(* IEC 61131-3 sources: std_i2980_v2.06_cp053/Source/IMM/ieccontrol/TIG, 14 files *)

(* ---- FArraySum.pu ---- *)
(*
@h    ! WARNING !
@h    The Kemro K2 system (including software) only meets category B according to EN 954-1,
@h    thus it is not intended for usage in safety-relevant control applications in the field
@h    of personal safety (e.g. emergency stop).
@h    To implement potentially necessary safety-relevant control tasks, always use additional
@h    external safety devices that are intended for the particular purpose, and meet the necessary
@h    functional safety.
@h    For further information see EN 954-1 (EN ISO 13849-1) and/or the K2-x00 user manual, chapter
@h    "CE conformity, directives and standards".

calculates sum of n arrayelements of type DINT
*)

IMPORT_OVER_LISTFILE
 tyTIGDInt

END_IMPORT

FUNCTION FArraySum : DINT #DUMMY_EDIT_BLOCK

VAR_INPUT
 iNumber : DINT (* number of array elements *);
END_VAR

VAR_IN_OUT
 array : tyTIGDInt (* array *);
END_VAR

VAR
 tmpSum : DINT;
 i : DINT;
END_VAR
#BEGIN_EDIT_BLOCK
(**************************************** WARNING ********************************************
 *** The KEBA Kemro K2 System including software is not intended for safety control tasks! ***
 ***                       For further information see Comment tab!                        ***
 *********************************************************************************************)

tmpSum := 0;

FOR i := 1 TO iNumber DO
   tmpSum := tmpSum + array[i];
END_FOR;

FArraySum:= tmpSum;

;#END_EDIT_BLOCK END_FUNCTION

#END_OF_IEC_PART

@Puma @IecEditor 6 60 @Pou 25
@@@BEG_Comment@@@
@h    ! WARNING !
@h    The Kemro K2 system (including software) only meets category B according to EN 954-1,
@h    thus it is not intended for usage in safety-relevant control applications in the field
@h    of personal safety (e.g. emergency stop).
@h    To implement potentially necessary safety-relevant control tasks, always use additional
@h    external safety devices that are intended for the particular purpose, and meet the necessary
@h    functional safety.
@h    For further information see EN 954-1 (EN ISO 13849-1) and/or the K2-x00 user manual, chapter
@h    "CE conformity, directives and standards".

calculates sum of n arrayelements of type DINT
@@@END_Comment@@@

@BEG_Contents

@BEG_Func
@RT(17)FuncTreeContainer
0
@END_Func

@BEG_Const
@RT(18)ConstTreeContainer
0
@END_Const

@BEG_Export

@BEG_Kind
@FUNCTION @RT(9)FArraySum @STRUCTURED_TEXT
@RT(4)DINT @RT(0) @RT(0)
@END_Kind

@BEG_Dcl
@RT(16)DclTreeContainer
4
@Var @RT(7)iNumber @RT(0) @T @F @DT @RT(4)DINT @RT(0) @T @T @BASIC 0 @F
@F @F
@T
@BEG_Attrib
3 @RT(0) @RT(24)number of array elements @RT(0)
@END_Attrib
1 1 @F @F @F @F

@Var @RT(5)array @RT(0) @T @T @DERIVED 0 @T @T @DT @RT(9)tyTIGDInt @RT(0) @T @T @UNKNOWN 0 @F
@F @F
@T
@BEG_Attrib
3 @RT(0) @RT(5)array @RT(0)
@END_Attrib
1 2 @F @F @F @F

@Var @RT(6)tmpSum @RT(0) @T @F @DT @RT(4)DINT @RT(0) @T @T @BASIC 0 @F
@F @F
@T
@BEG_Attrib
3 @RT(0) @RT(0) @RT(0)
@END_Attrib
1 0 @F @F @F @F

@Var @RT(1)i @RT(0) @T @F @DT @RT(4)DINT @RT(0) @T @T @BASIC 0 @F
@F @F
@T
@BEG_Attrib
3 @RT(0) @RT(0) @RT(0)
@END_Attrib
1 0 @F @F @F @F

@END_Dcl

@END_Export

@BEG_Body
@TL(13)
(**************************************** WARNING ********************************************
 *** The KEBA Kemro K2 System including software is not intended for safety control tasks! ***
 ***                       For further information see Comment tab!                        ***
 *********************************************************************************************)

tmpSum := 0;

FOR i := 1 TO iNumber DO
   tmpSum := tmpSum + array[i];
END_FOR;

FArraySum:= tmpSum;

@END_Body

@END_Contents

(* ---- FDeleteActDSFiles.pu ---- *)
(*
@h    ! WARNING !
@h    The Kemro K2 system (including software) only meets category B according to EN 954-1,
@h    thus it is not intended for usage in safety-relevant control applications in the field
@h    of personal safety (e.g. emergency stop).
@h    To implement potentially necessary safety-relevant control tasks, always use additional
@h    external safety devices that are intended for the particular purpose, and meet the necessary
@h    functional safety.
@h    For further information see EN 954-1 (EN ISO 13849-1) and/or the K2-x00 user manual, chapter
@h    "CE conformity, directives and standards".

deletes and creates temporary directory for datasettransfer to tig

@FunctionID: A-VAR-14
@FunctionID: A-VAR-15
TIG 3.10
*)

IMPORT_OVER_LISTFILE
 KFILE_Status

END_IMPORT

FUNCTION FDeleteActDSFiles : BOOL #DUMMY_EDIT_BLOCK

VAR_IN_OUT
 sPath : STRING(255);
END_VAR

VAR
 s : KFILE_Status;
END_VAR
#BEGIN_EDIT_BLOCK
(**************************************** WARNING ********************************************
 *** The KEBA Kemro K2 System including software is not intended for safety control tasks! ***
 ***                       For further information see Comment tab!                        ***
 *********************************************************************************************)

s := KFILE_RemoveDir(sPath);
s := KFILE_MakeDir(sPath);
FDeleteActDSFiles := TRUE;

;#END_EDIT_BLOCK END_FUNCTION

#END_OF_IEC_PART

@Puma @IecEditor 6 60 @Pou 25
@@@BEG_Comment@@@
@h    ! WARNING !
@h    The Kemro K2 system (including software) only meets category B according to EN 954-1,
@h    thus it is not intended for usage in safety-relevant control applications in the field
@h    of personal safety (e.g. emergency stop).
@h    To implement potentially necessary safety-relevant control tasks, always use additional
@h    external safety devices that are intended for the particular purpose, and meet the necessary
@h    functional safety.
@h    For further information see EN 954-1 (EN ISO 13849-1) and/or the K2-x00 user manual, chapter
@h    "CE conformity, directives and standards".

deletes and creates temporary directory for datasettransfer to tig

@FunctionID: A-VAR-14
@FunctionID: A-VAR-15
TIG 3.10
@@@END_Comment@@@

@BEG_Contents

@BEG_Func
@RT(17)FuncTreeContainer
0
@END_Func

@BEG_Const
@RT(18)ConstTreeContainer
0
@END_Const

@BEG_Export

@BEG_Kind
@FUNCTION @RT(17)FDeleteActDSFiles @STRUCTURED_TEXT
@RT(4)BOOL @RT(0) @RT(0)
@END_Kind

@BEG_Dcl
@RT(16)DclTreeContainer
2
@Var @RT(5)sPath @RT(0) @T @F @DT @RT(11)STRING(255) @RT(0) @T @T @STRING 0 @F @RT(3)255 @F
@F @F
@T
@BEG_Attrib
3 @RT(0) @RT(0) @RT(0)
@END_Attrib
1 2 @F @F @F @F

@Var @RT(1)s @RT(0) @T @T @DERIVED 0 @T @T @DT @RT(12)KFILE_Status @RT(0) @T @T @UNKNOWN 0 @F
@F @F
@T
@BEG_Attrib
3 @RT(0) @RT(0) @RT(0)
@END_Attrib
1 0 @F @F @F @F

@END_Dcl

@END_Export

@BEG_Body
@TL(9)
(**************************************** WARNING ********************************************
 *** The KEBA Kemro K2 System including software is not intended for safety control tasks! ***
 ***                       For further information see Comment tab!                        ***
 *********************************************************************************************)

s := KFILE_RemoveDir(sPath);
s := KFILE_MakeDir(sPath);
FDeleteActDSFiles := TRUE;

@END_Body

@END_Contents

(* ---- FBHmiDataSet.pu ---- *)
(*
@h    ! WARNING !
@h    The Kemro K2 system (including software) only meets category B according to EN 954-1,
@h    thus it is not intended for usage in safety-relevant control applications in the field
@h    of personal safety (e.g. emergency stop).
@h    To implement potentially necessary safety-relevant control tasks, always use additional
@h    external safety devices that are intended for the particular purpose, and meet the necessary
@h    functional safety.
@h    For further information see EN 954-1 (EN ISO 13849-1) and/or the K2-x00 user manual, chapter
@h    "CE conformity, directives and standards".

command to HMI: load or save dataset

@FunctionID: A-VAR-16.5
TIG 3.11.6
*)

IMPORT_OVER_LISTFILE
 tsTIGHmi
, R_TRIG

END_IMPORT

FUNCTION_BLOCK FBHmiDataSet #DUMMY_EDIT_BLOCK

VAR_INPUT
 Execute : BOOL (* starts command to hmi *);
 Save : BOOL (* false ... LOAD, true ... SAVE *);
END_VAR

VAR_IN_OUT
 sParam : STRING(255) (* name of dataset *);
END_VAR

VAR_OUTPUT
 Done : BOOL (* command done without error *);
 Error : BOOL (* command done but error *);
END_VAR

SYSTEM_VAR
 sv_TIGHmi : tsTIGHmi;
END_VAR

VAR
 fbExecTrig : R_TRIG;
 miStart : INT;
 bStarted : BOOL;
END_VAR
#BEGIN_EDIT_BLOCK
(**************************************** WARNING ********************************************
 *** The KEBA Kemro K2 System including software is not intended for safety control tasks! ***
 ***                       For further information see Comment tab!                        ***
 *********************************************************************************************)

fbExecTrig(Execute);

IF Execute = FALSE THEN
   Done := FALSE;
   Error := FALSE;
END_IF;

IF NOT bStarted THEN
   IF fbExecTrig.Q THEN
      bStarted := TRUE;
      miStart := DINT_TO_INT(sv_TIGHmi.dataSet.DSCmd2Hmi.iCmd);

      sv_TIGHmi.dataSet.DSCmd2Hmi.sParam := sParam;

      // miStart MOD 2 = 1 starts the command
      miStart := miStart + ((miStart MOD 2) + 1);

      sv_TIGHmi.dataSet.DSCmd2Hmi.iCmd := DWORD_TO_DINT(SHL(BOOL_TO_DWORD(Save), 16)) + INT_TO_DINT(miStart);
   END_IF;
ELSE
   // MOD 2 = 0 cmd finished
   IF (sv_TIGHmi.dataSet.DSCmd2Hmi.iCmd MOD 2) = 0 THEN
      bStarted := FALSE;
      Error := DWORD_TO_BOOL((DINT_TO_DWORD(sv_TIGHmi.dataSet.DSCmd2Hmi.iCmd) AND 16#FFFF0000));
      Done := NOT Error;
   END_IF;
END_IF;

;#END_EDIT_BLOCK END_FUNCTION_BLOCK

#END_OF_IEC_PART

@Puma @IecEditor 6 60 @Pou 25
@@@BEG_Comment@@@
@h    ! WARNING !
@h    The Kemro K2 system (including software) only meets category B according to EN 954-1,
@h    thus it is not intended for usage in safety-relevant control applications in the field
@h    of personal safety (e.g. emergency stop).
@h    To implement potentially necessary safety-relevant control tasks, always use additional
@h    external safety devices that are intended for the particular purpose, and meet the necessary
@h    functional safety.
@h    For further information see EN 954-1 (EN ISO 13849-1) and/or the K2-x00 user manual, chapter
@h    "CE conformity, directives and standards".

command to HMI: load or save dataset

@FunctionID: A-VAR-16.5
TIG 3.11.6
@@@END_Comment@@@

@BEG_Contents

@BEG_Func
@RT(17)FuncTreeContainer
0
@END_Func

@BEG_Const
@RT(18)ConstTreeContainer
0
@END_Const

@BEG_Export

@BEG_Kind
@FUNCTION_BLOCK @RT(12)FBHmiDataSet @STRUCTURED_TEXT
@RT(0) @RT(0) @RT(0)
@END_Kind

@BEG_Dcl
@RT(16)DclTreeContainer
9
@Var @RT(9)sv_TIGHmi @RT(0) @T @T @DERIVED 0 @T @T @DT @RT(8)tsTIGHmi @RT(0) @T @T @UNKNOWN 0 @F
@F @F
@T
@BEG_Attrib
3 @RT(0) @RT(0) @RT(0)
@END_Attrib
1 8 @F @F @F @F

@Var @RT(7)Execute @RT(0) @T @F @DT @RT(4)BOOL @RT(0) @T @T @BASIC 0 @F
@F @F
@T
@BEG_Attrib
3 @RT(0) @RT(21)starts command to hmi @RT(0)
@END_Attrib
1 1 @F @F @F @F

@Var @RT(4)Save @RT(0) @T @F @DT @RT(4)BOOL @RT(0) @T @T @BASIC 0 @F
@F @F
@T
@BEG_Attrib
3 @RT(0) @RT(29)false ... LOAD, true ... SAVE @RT(0)
@END_Attrib
1 1 @F @F @F @F

@Var @RT(6)sParam @RT(0) @T @F @DT @RT(11)STRING(255) @RT(0) @T @T @STRING 0 @F @RT(3)255 @F
@F @F
@T
@BEG_Attrib
3 @RT(0) @RT(15)name of dataset @RT(0)
@END_Attrib
1 2 @F @F @F @F

@Var @RT(4)Done @RT(0) @T @F @DT @RT(4)BOOL @RT(0) @T @T @BASIC 0 @F
@F @F
@T
@BEG_Attrib
3 @RT(0) @RT(26)command done without error @RT(0)
@END_Attrib
1 3 @F @F @F @F

@Var @RT(5)Error @RT(0) @T @F @DT @RT(4)BOOL @RT(0) @T @T @BASIC 0 @F
@F @F
@T
@BEG_Attrib
3 @RT(0) @RT(22)command done but error @RT(0)
@END_Attrib
1 3 @F @F @F @F

@Var @RT(10)fbExecTrig @RT(0) @T @T @DERIVED 0 @T @T @DT @RT(6)R_TRIG @RT(0) @T @T @UNKNOWN 0 @F
@F @F
@T
@BEG_Attrib
3 @RT(0) @RT(0) @RT(0)
@END_Attrib
1 0 @F @F @F @F

@Var @RT(7)miStart @RT(0) @T @F @DT @RT(3)INT @RT(0) @T @T @BASIC 0 @F
@F @F
@T
@BEG_Attrib
3 @RT(0) @RT(0) @RT(0)
@END_Attrib
1 0 @F @F @F @F

@Var @RT(8)bStarted @RT(0) @T @F @DT @RT(4)BOOL @RT(0) @T @T @BASIC 0 @F
@F @F
@T
@BEG_Attrib
3 @RT(0) @RT(0) @RT(0)
@END_Attrib
1 0 @F @F @F @F

@END_Dcl

@END_Export

@BEG_Body
@TL(33)
(**************************************** WARNING ********************************************
 *** The KEBA Kemro K2 System including software is not intended for safety control tasks! ***
 ***                       For further information see Comment tab!                        ***
 *********************************************************************************************)

fbExecTrig(Execute);

IF Execute = FALSE THEN
   Done := FALSE;
   Error := FALSE;
END_IF;

IF NOT bStarted THEN
   IF fbExecTrig.Q THEN
      bStarted := TRUE;
      miStart := DINT_TO_INT(sv_TIGHmi.dataSet.DSCmd2Hmi.iCmd);

      sv_TIGHmi.dataSet.DSCmd2Hmi.sParam := sParam;

      // miStart MOD 2 = 1 starts the command
      miStart := miStart + ((miStart MOD 2) + 1);

      sv_TIGHmi.dataSet.DSCmd2Hmi.iCmd := DWORD_TO_DINT(SHL(BOOL_TO_DWORD(Save), 16)) + INT_TO_DINT(miStart);
   END_IF;
ELSE
   // MOD 2 = 0 cmd finished
   IF (sv_TIGHmi.dataSet.DSCmd2Hmi.iCmd MOD 2) = 0 THEN
      bStarted := FALSE;
      Error := DWORD_TO_BOOL((DINT_TO_DWORD(sv_TIGHmi.dataSet.DSCmd2Hmi.iCmd) AND 16#FFFF0000));
      Done := NOT Error;
   END_IF;
END_IF;

@END_Body

@END_Contents

(* ---- ABCavities.pu ---- *)
(*
@h    ! WARNING !
@h    The Kemro K2 system (including software) only meets category B according to EN 954-1,
@h    thus it is not intended for usage in safety-relevant control applications in the field
@h    of personal safety (e.g. emergency stop).
@h    To implement potentially necessary safety-relevant control tasks, always use additional
@h    external safety devices that are intended for the particular purpose, and meet the necessary
@h    functional safety.
@h    For further information see EN 954-1 (EN ISO 13849-1) and/or the K2-x00 user manual, chapter
@h    "CE conformity, directives and standards".

assignment articles to cavities

@FunctionID: A-Mask-7

*)

IMPORT_OVER_LISTFILE
 cNoMaxArticles
, tsTIGHmi
, tsTIG

END_IMPORT

ALGORITHM_BLOCK ABCavities #DUMMY_EDIT_BLOCK

SYSTEM_VAR
 sv_TIGHmi : tsTIGHmi;
 sv_TIG : tsTIG;
END_VAR

SYSTEM_OBJECT
 TaskVis : TASK;
END_OBJECT

(*
@h    ! WARNING !
@h    The Kemro K2 system (including software) only meets category B according to EN 954-1,
@h    thus it is not intended for usage in safety-relevant control applications in the field
@h    of personal safety (e.g. emergency stop).
@h    To implement potentially necessary safety-relevant control tasks, always use additional
@h    external safety devices that are intended for the particular purpose, and meet the necessary
@h    functional safety.
@h    For further information see EN 954-1 (EN ISO 13849-1) and/or the K2-x00 user manual, chapter
@h    "CE conformity, directives and standards".

block initialisation

@FunctionID: A-MASK-7

*)

ALGORITHM aInit

#BEGIN_EDIT_BLOCK
(**************************************** WARNING ********************************************
 *** The KEBA Kemro K2 System including software is not intended for safety control tasks! ***
 ***                       For further information see Comment tab!                        ***
 *********************************************************************************************)

;#END_EDIT_BLOCK END_ALGORITHM

(*
@h    ! WARNING !
@h    The Kemro K2 system (including software) only meets category B according to EN 954-1,
@h    thus it is not intended for usage in safety-relevant control applications in the field
@h    of personal safety (e.g. emergency stop).
@h    To implement potentially necessary safety-relevant control tasks, always use additional
@h    external safety devices that are intended for the particular purpose, and meet the necessary
@h    functional safety.
@h    For further information see EN 954-1 (EN ISO 13849-1) and/or the K2-x00 user manual, chapter
@h    "CE conformity, directives and standards".

@FunctionID: A-Mask-7

*)

POSTUPDATE_ALGORITHM aSetCavities ON TaskVis WITH sv_TIG.productionData.Set.yCavity

VAR_TEMP
 i : DINT;
END_VAR
#BEGIN_EDIT_BLOCK
(**************************************** WARNING ********************************************
 *** The KEBA Kemro K2 System including software is not intended for safety control tasks! ***
 ***                       For further information see Comment tab!                        ***
 *********************************************************************************************)

FOR i:=1 TO 32 DO
   sv_TIGHmi.productionData.cavities.ActCavSelected[i] := TRUE;
END_FOR;
sv_TIG.productionData.Act.yCavity := sv_TIG.productionData.Set.yCavity;
sv_TIGHmi.productionData.cavities.iSetCavChanged := sv_TIGHmi.productionData.cavities.iSetCavChanged + 1;

;#END_EDIT_BLOCK END_ALGORITHM

(*
@h    ! WARNING !
@h    The Kemro K2 system (including software) only meets category B according to EN 954-1,
@h    thus it is not intended for usage in safety-relevant control applications in the field
@h    of personal safety (e.g. emergency stop).
@h    To implement potentially necessary safety-relevant control tasks, always use additional
@h    external safety devices that are intended for the particular purpose, and meet the necessary
@h    functional safety.
@h    For further information see EN 954-1 (EN ISO 13849-1) and/or the K2-x00 user manual, chapter
@h    "CE conformity, directives and standards".

@FunctionID: A-Mask-7

*)

POSTUPDATE_ALGORITHM pActSelChanged ON TaskVis WITH sv_TIGHmi.productionData.cavities.ActCavSelected

VAR_TEMP
 i : DINT;
 k : DINT;
END_VAR

VAR
 n : DINT;
 m : DINT;
END_VAR
#BEGIN_EDIT_BLOCK
(**************************************** WARNING ********************************************
 *** The KEBA Kemro K2 System including software is not intended for safety control tasks! ***
 ***                       For further information see Comment tab!                        ***
 *********************************************************************************************)

m := 0;
FOR k := 1 TO cNoMaxArticles DO
  n := 0;
  FOR i := 1 TO sv_TIG.productionData.Set.yCavity[k] DO
    m := m + 1;
    n := n + BOOL_TO_DINT(sv_TIGHmi.productionData.cavities.ActCavSelected[m]);
  END_FOR;
  sv_TIG.productionData.Act.yCavity[k] := n;
END_FOR;

;#END_EDIT_BLOCK END_ALGORITHM

END_ALGORITHM_BLOCK

#END_OF_IEC_PART

@Puma @IecEditor 6 68 @Pou 25
@@@BEG_Comment@@@
@h    ! WARNING !
@h    The Kemro K2 system (including software) only meets category B according to EN 954-1,
@h    thus it is not intended for usage in safety-relevant control applications in the field
@h    of personal safety (e.g. emergency stop).
@h    To implement potentially necessary safety-relevant control tasks, always use additional
@h    external safety devices that are intended for the particular purpose, and meet the necessary
@h    functional safety.
@h    For further information see EN 954-1 (EN ISO 13849-1) and/or the K2-x00 user manual, chapter
@h    "CE conformity, directives and standards".

assignment articles to cavities

@FunctionID: A-Mask-7

@@@END_Comment@@@

@BEG_Contents

@BEG_Func
@RT(17)FuncTreeContainer
0
@END_Func

@BEG_Const
@RT(18)ConstTreeContainer
1
@Var @RT(14)cNoMaxArticles @RT(0) @T @F @DT @RT(0) @RT(0) @T @T @UNKNOWN 0 @F
@F @F
@T
@BEG_Attrib
0 @RT(0) @RT(0)
@END_Attrib
1 1 @F @F @F @F

@END_Const

@BEG_Export

@BEG_Kind
@ALGORITHM_BLOCK @RT(10)ABCavities @STRUCTURED_TEXT
@RT(0) @RT(0) @RT(0)
@END_Kind

@BEG_Dcl
@RT(16)DclTreeContainer
3
@Var @RT(9)sv_TIGHmi @RT(0) @T @T @DERIVED 0 @T @T @DT @RT(8)tsTIGHmi @RT(0) @T @T @UNKNOWN 0 @F
@F @F
@T
@BEG_Attrib
3 @RT(0) @RT(0) @RT(0)
@END_Attrib
1 8 @F @F @F @F

@Var @RT(6)sv_TIG @RT(0) @T @T @DERIVED 0 @T @T @DT @RT(5)tsTIG @RT(0) @T @T @UNKNOWN 0 @F
@F @F
@T
@BEG_Attrib
3 @RT(0) @RT(0) @RT(0)
@END_Attrib
1 8 @F @F @F @F

@Var @RT(7)TaskVis @RT(0) @T @F @DT @RT(4)TASK @RT(0) @T @T @BASIC 0 @F
@F @F
@T
@BEG_Attrib
3 @RT(0) @RT(0) @RT(0)
@END_Attrib
1 7 @F @F @F @F

@END_Dcl

@END_Export

@BEG_Body

3

@BEG_Export

@BEG_Algo
@ALGORITHM @RT(5)aInit @STRUCTURED_TEXT
@RT(0) @RT(0) @RT(0) @F @F
@END_Algo

@BEG_Dcl
@RT(16)DclTreeContainer
0
@END_Dcl

@END_Export

@BEG_Export

@BEG_Algo
@POSTUPDATE_ALGORITHM @RT(12)aSetCavities @STRUCTURED_TEXT
@RT(0) @RT(33)sv_TIG.productionData.Set.yCavity @RT(7)TaskVis @F @F
@END_Algo

@BEG_Dcl
@RT(16)DclTreeContainer
1
@Var @RT(1)i @RT(0) @T @F @DT @RT(4)DINT @RT(0) @T @T @BASIC 0 @F
@F @F
@T
@BEG_Attrib
3 @RT(0) @RT(0) @RT(0)
@END_Attrib
1 4 @F @F @F @F

@END_Dcl

@END_Export

@BEG_Export

@BEG_Algo
@POSTUPDATE_ALGORITHM @RT(14)pActSelChanged @STRUCTURED_TEXT
@RT(0) @RT(48)sv_TIGHmi.productionData.cavities.ActCavSelected @RT(7)TaskVis @F @F
@END_Algo

@BEG_Dcl
@RT(16)DclTreeContainer
4
@Var @RT(1)i @RT(0) @T @F @DT @RT(4)DINT @RT(0) @T @T @BASIC 0 @F
@F @F
@T
@BEG_Attrib
3 @RT(0) @RT(0) @RT(0)
@END_Attrib
1 4 @F @F @F @F

@Var @RT(1)k @RT(0) @T @F @DT @RT(4)DINT @RT(0) @T @T @BASIC 0 @F
@F @F
@T
@BEG_Attrib
3 @RT(0) @RT(0) @RT(0)
@END_Attrib
1 4 @F @F @F @F

@Var @RT(1)n @RT(0) @T @F @DT @RT(4)DINT @RT(0) @T @T @BASIC 0 @F
@F @F
@T
@BEG_Attrib
3 @RT(0) @RT(0) @RT(0)
@END_Attrib
1 0 @F @F @F @F

@Var @RT(1)m @RT(0) @T @F @DT @RT(4)DINT @RT(0) @T @T @BASIC 0 @F
@F @F
@T
@BEG_Attrib
3 @RT(0) @RT(0) @RT(0)
@END_Attrib
1 0 @F @F @F @F

@END_Dcl

@END_Export

@BEG_Body
@TL(6)
(**************************************** WARNING ********************************************
 *** The KEBA Kemro K2 System including software is not intended for safety control tasks! ***
 ***                       For further information see Comment tab!                        ***
 *********************************************************************************************)

@END_Body

@@@BEG_Comment@@@
@TL(14)
@h    ! WARNING !
@h    The Kemro K2 system (including software) only meets category B according to EN 954-1,
@h    thus it is not intended for usage in safety-relevant control applications in the field
@h    of personal safety (e.g. emergency stop).
@h    To implement potentially necessary safety-relevant control tasks, always use additional
@h    external safety devices that are intended for the particular purpose, and meet the necessary
@h    functional safety.
@h    For further information see EN 954-1 (EN ISO 13849-1) and/or the K2-x00 user manual, chapter
@h    "CE conformity, directives and standards".

block initialisation

@FunctionID: A-MASK-7

@@@END_Comment@@@

@BEG_Body
@TL(13)
(**************************************** WARNING ********************************************
 *** The KEBA Kemro K2 System including software is not intended for safety control tasks! ***
 ***                       For further information see Comment tab!                        ***
 *********************************************************************************************)

FOR i:=1 TO 32 DO
   sv_TIGHmi.productionData.cavities.ActCavSelected[i] := TRUE;
END_FOR;
sv_TIG.productionData.Act.yCavity := sv_TIG.productionData.Set.yCavity;
sv_TIGHmi.productionData.cavities.iSetCavChanged := sv_TIGHmi.productionData.cavities.iSetCavChanged + 1;

@END_Body

@@@BEG_Comment@@@
@TL(14)
@h    ! WARNING !
@h    The Kemro K2 system (including software) only meets category B according to EN 954-1,
@h    thus it is not intended for usage in safety-relevant control applications in the field
@h    of personal safety (e.g. emergency stop).
@h    To implement potentially necessary safety-relevant control tasks, always use additional
@h    external safety devices that are intended for the particular purpose, and meet the necessary
@h    functional safety.
@h    For further information see EN 954-1 (EN ISO 13849-1) and/or the K2-x00 user manual, chapter
@h    "CE conformity, directives and standards".

@FunctionID: A-Mask-7

@@@END_Comment@@@

@BEG_Body
@TL(19)
(**************************************** WARNING ********************************************
 *** The KEBA Kemro K2 System including software is not intended for safety control tasks! ***
 ***                       For further information see Comment tab!                        ***
 *********************************************************************************************)

m := 0;
FOR k := 1 TO cNoMaxArticles DO
  n := 0;
  FOR i := 1 TO sv_TIG.productionData.Set.yCavity[k] DO
    m := m + 1;
    n := n + BOOL_TO_DINT(sv_TIGHmi.productionData.cavities.ActCavSelected[m]);
  END_FOR;
  sv_TIG.productionData.Act.yCavity[k] := n;
END_FOR;

@END_Body

@@@BEG_Comment@@@
@TL(14)
@h    ! WARNING !
@h    The Kemro K2 system (including software) only meets category B according to EN 954-1,
@h    thus it is not intended for usage in safety-relevant control applications in the field
@h    of personal safety (e.g. emergency stop).
@h    To implement potentially necessary safety-relevant control tasks, always use additional
@h    external safety devices that are intended for the particular purpose, and meet the necessary
@h    functional safety.
@h    For further information see EN 954-1 (EN ISO 13849-1) and/or the K2-x00 user manual, chapter
@h    "CE conformity, directives and standards".

@FunctionID: A-Mask-7

@@@END_Comment@@@
@END_Body

@END_Contents
